{attribute 'GeneratedUsingTerminal: EL9576-0000-0020'}
{attribute addProperty BoxType "EL9576-0000-0020"}
{attribute addProperty Description "EL9576 Brake chopper terminal"}
{attribute addProperty Physics "KK"}
{attribute addProperty Id "BCT_InputsAT %I*BCT_Inputs_8B1D510C16WcStateAT %I*WcState_9091E0EB2InfoDataAT %I*InfoData_32EB74EA10"}
{attribute addProperty CRC "270005413"}
{attribute addProperty Size "28"}
TYPE EL9576_1017F4A5 EXTENDS EtcSlaveTerminalBase_947E5A46 :
STRUCT
	{attribute addProperty Name "BCT_Inputs"}
	BCT_Inputs : BCT_Inputs_8B1D510C;
	{attribute addProperty Name "WcState"}
	WcState : WcState_9091E0EB;
	{attribute addProperty Name "InfoData"}
	InfoData : InfoData_32EB74EA;
END_STRUCT
END_TYPE

(* stored: Version 1.2.0.0, ProductVersion 3.1.4024.9
   DUT EL9576_1017F4A5: Id {e438c0b9-7a0b-4f6e-a3d8-b8e107d0310a} *)
